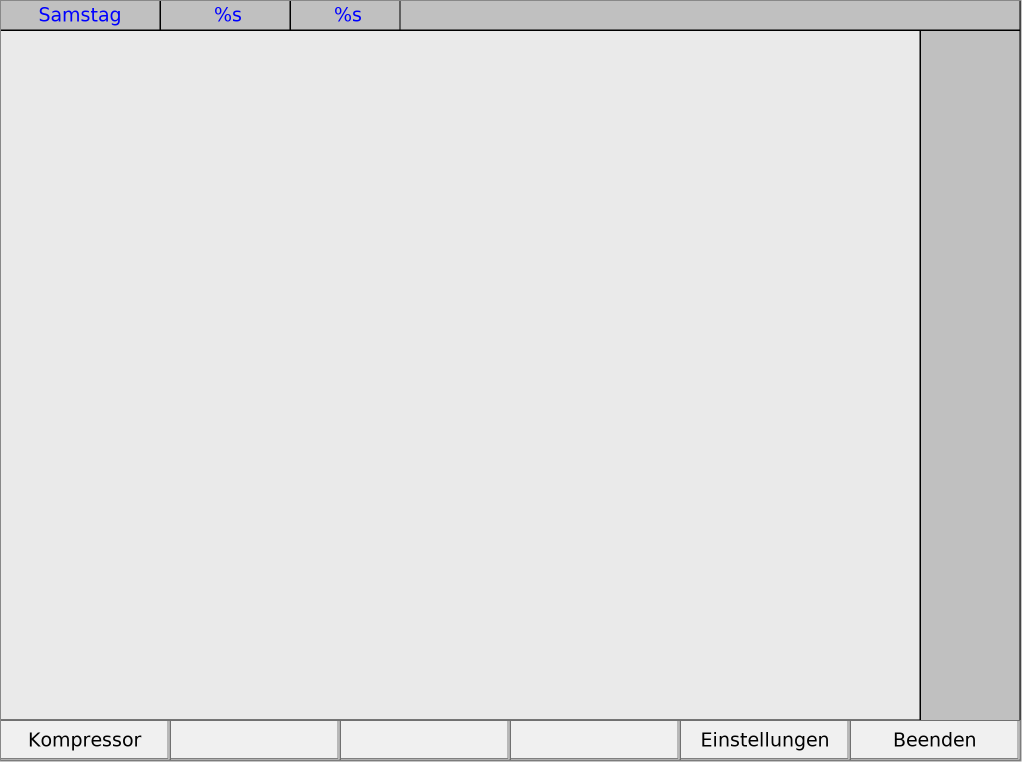
VISUALIZATION V_Main_PC  // 1022x762
    Rectangle (920,30 100x730)
    Rectangle (0,0 1020x30)
    Rectangle (0,30 920x690)
    Rectangle (0,720 1020x40)
    Rectangle (160,0 130x30), "%s", text variable: gfbSystemCX.OUTszDate
    Rectangle (290,0 110x30), "%s", text variable: gfbSystemCX.OUTszClock
    Button (850,720 170x40), "Beenden"
    Button (680,720 170x40), "Einstellungen"
        OnMouseUp: change screen: V_Einstellungen
    Button (510,720 170x40)
    Button (340,720 170x40)
    Button (170,720 170x40)
    Button (0,720 170x40), "Kompressor"
        OnMouseClick: change screen: V_KomprWRG
        OnMouseUp: change screen: V_KomprWRG
    Rectangle (0,0 160x30), "Sonntag", invisible if: gfbSystemCX.OUTeDayOfWeek > 0
    Rectangle (0,0 160x30), "Montag", invisible if: gfbSystemCX.OUTeDayOfWeek <> 1
    Rectangle (0,0 160x30), "Dienstag", invisible if: gfbSystemCX.OUTeDayOfWeek <> 2
    Rectangle (0,0 160x30), "Mittwoch", invisible if: gfbSystemCX.OUTeDayOfWeek <> 3
    Rectangle (0,0 160x30), "Donnerstag", invisible if: gfbSystemCX.OUTeDayOfWeek <> 4
    Rectangle (0,0 160x30), "Freitag", invisible if: gfbSystemCX.OUTeDayOfWeek <> 5
    Rectangle (0,0 160x30), "Samstag", invisible if: gfbSystemCX.OUTeDayOfWeek <> 6
END_VISUALIZATION

(* stored: Version 1.1.0.1, ProductVersion 3.1.4018.9
   Visu V_Main_PC: Id {91c9f370-eadf-4c5d-89a8-1a6c498e4233} *)
